Omron CX-Programmer project NewProject (CX-Programmer 9.61)

# PLC NewPLC1: CP1H XA

## Global symbols (name address type ; comment)
0.01 BOOL  ; Gr_out_up
0.02 BOOL  ; up_outside_1
0.03 BOOL  ; dn_outside_1
0.04 BOOL  ; dn_outside_2
0.05 BOOL  ; Gr_inside
0.06 BOOL  ; 1_inside
0.07 BOOL  ; 2_inside
100.01 BOOL  ; Motorup
100.02 BOOL  ; Motordown
100.03 BOOL  ; slow
100.04 BOOL  ; D_open
100.05 BOOL  ; D_close
100.09 BOOL  ; M111
10.00 BOOL  ; M1
10.01 BOOL  ; M2
10.02 BOOL  ; M3
10.03 BOOL  ; M4
10.04 BOOL  ; M5
10.05 BOOL  ; M3
10.06 BOOL  ; M7
10.07 BOOL  ; M8
10.08 BOOL  ; M9
10.09 BOOL  ; M10
10.10 BOOL  ; M11
10.11 BOOL  ; M12
10.12 BOOL  ; M13
10.13 BOOL  ; G_motor_up
10.14 BOOL  ; G_motorup_slow
10.15 BOOL  ; 1F_motor_up
11.01 BOOL  ; 1F_motor_slow
11.02 BOOL  ; 2F_motor_down
11.03 BOOL  ; 2F_motor_slow
11.04 BOOL  ; 1F_motor_down
11.05 BOOL  ; 1F_motor_slow
11.06 BOOL  ; G_motor_up_to_2nd
11.07 BOOL  ; G_motor_slow_to_2nd
11.08 BOOL  ; 2F_motor_down_toGround
11.09 BOOL  ; 2F_motor_slow_toGround
12.01 BOOL  ; 1F_pressed_slow
12.02 BOOL  ; 1F_pressed_stop
12.03 BOOL  ; 1F_pressed_slow1
12.04 BOOL  ; 1F_pressed_stopp
12.05 BOOL  ; M_2inside
12.06 BOOL  ; M_Ginside
13.01 BOOL  ; D_Open_for_outside
13.02 BOOL  ; D_Close_for_outside
13.03 BOOL  ; D_open_for_inside
13.04 BOOL  ; D_close_for_inside
13.05 BOOL  ; D_close_memory
13.06 BOOL  ; D_close_memory1
14.01 BOOL  ; MD1
14.02 BOOL  ; MD2
14.03 BOOL  ; MD3
14.04 BOOL  ; MD4
15.01 BOOL  ; M111
1.01 BOOL  ; LS0
1.02 BOOL  ; LS0(High)
1.03 BOOL  ; LS1
1.04 BOOL  ; LS1(High)
1.05 BOOL  ; LS2
1.06 BOOL  ; LS1(Low)
1.07 BOOL  ; LS0(Low)
T0000 BOOL  ; T1
T0001 BOOL  ; T2
T0002 BOOL  ; T3
T0003 BOOL  ; T4

## Program NewProgram1 (cyclic task 0)

### Section Section1

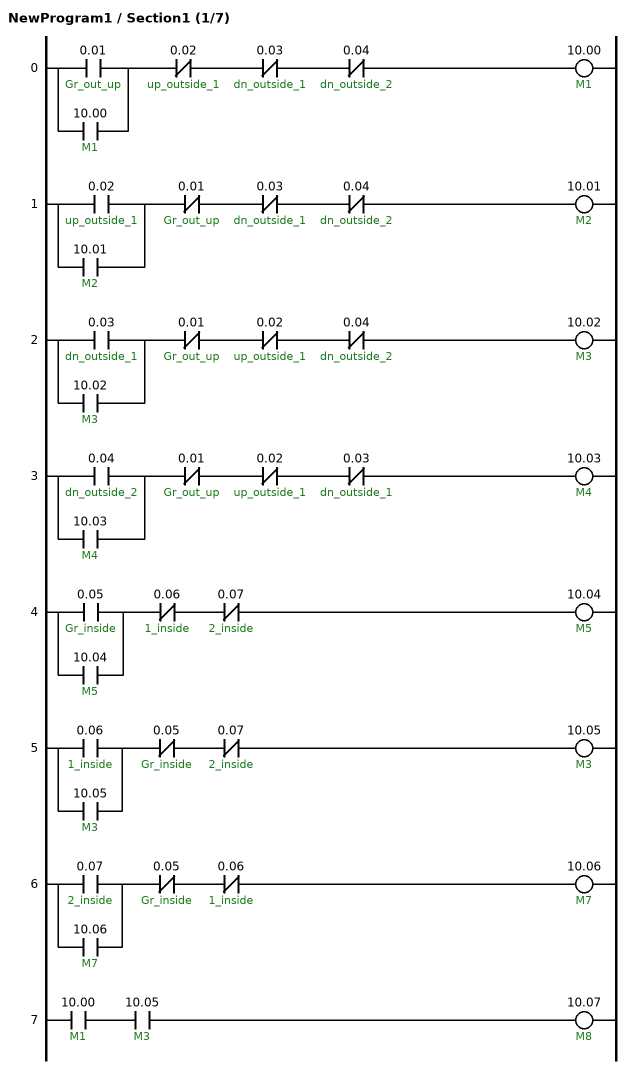
; rung 0
LD 0.01  ; Gr_out_up
OR 10.00  ; M1
ANDNOT 0.02  ; up_outside_1
ANDNOT 0.03  ; dn_outside_1
ANDNOT 0.04  ; dn_outside_2
OUT 10.00  ; M1
; rung 1
LD 0.02  ; up_outside_1
OR 10.01  ; M2
ANDNOT 0.01  ; Gr_out_up
ANDNOT 0.03  ; dn_outside_1
ANDNOT 0.04  ; dn_outside_2
OUT 10.01  ; M2
; rung 2
LD 0.03  ; dn_outside_1
OR 10.02  ; M3
ANDNOT 0.01  ; Gr_out_up
ANDNOT 0.02  ; up_outside_1
ANDNOT 0.04  ; dn_outside_2
OUT 10.02  ; M3
; rung 3
LD 0.04  ; dn_outside_2
OR 10.03  ; M4
ANDNOT 0.01  ; Gr_out_up
ANDNOT 0.02  ; up_outside_1
ANDNOT 0.03  ; dn_outside_1
OUT 10.03  ; M4
; rung 4
LD 0.05  ; Gr_inside
OR 10.04  ; M5
ANDNOT 0.06  ; 1_inside
ANDNOT 0.07  ; 2_inside
OUT 10.04  ; M5
; rung 5
LD 0.06  ; 1_inside
OR 10.05  ; M3
ANDNOT 0.05  ; Gr_inside
ANDNOT 0.07  ; 2_inside
OUT 10.05  ; M3
; rung 6
LD 0.07  ; 2_inside
OR 10.06  ; M7
ANDNOT 0.05  ; Gr_inside
ANDNOT 0.06  ; 1_inside
OUT 10.06  ; M7
; rung 7
LD 10.00  ; M1
AND 10.05  ; M3
OUT 10.07  ; M8

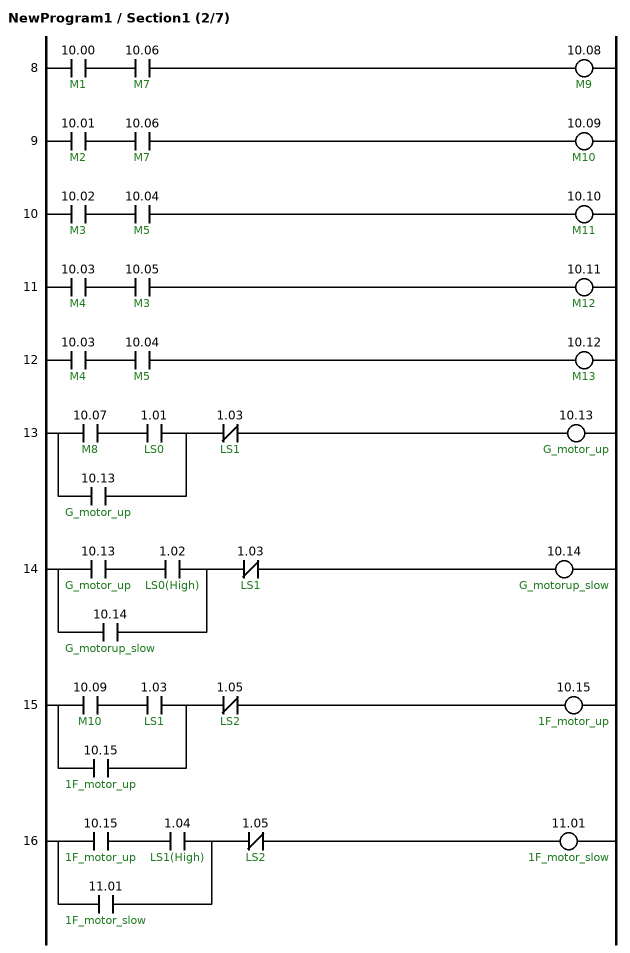
; rung 8
LD 10.00  ; M1
AND 10.06  ; M7
OUT 10.08  ; M9
; rung 9
LD 10.01  ; M2
AND 10.06  ; M7
OUT 10.09  ; M10
; rung 10
LD 10.02  ; M3
AND 10.04  ; M5
OUT 10.10  ; M11
; rung 11
LD 10.03  ; M4
AND 10.05  ; M3
OUT 10.11  ; M12
; rung 12
LD 10.03  ; M4
AND 10.04  ; M5
OUT 10.12  ; M13
; rung 13
LD 10.07  ; M8
AND 1.01  ; LS0
OR 10.13  ; G_motor_up
ANDNOT 1.03  ; LS1
OUT 10.13  ; G_motor_up
; rung 14
LD 10.13  ; G_motor_up
AND 1.02  ; LS0(High)
OR 10.14  ; G_motorup_slow
ANDNOT 1.03  ; LS1
OUT 10.14  ; G_motorup_slow
; rung 15
LD 10.09  ; M10
AND 1.03  ; LS1
OR 10.15  ; 1F_motor_up
ANDNOT 1.05  ; LS2
OUT 10.15  ; 1F_motor_up
; rung 16
LD 10.15  ; 1F_motor_up
AND 1.04  ; LS1(High)
OR 11.01  ; 1F_motor_slow
ANDNOT 1.05  ; LS2
OUT 11.01  ; 1F_motor_slow

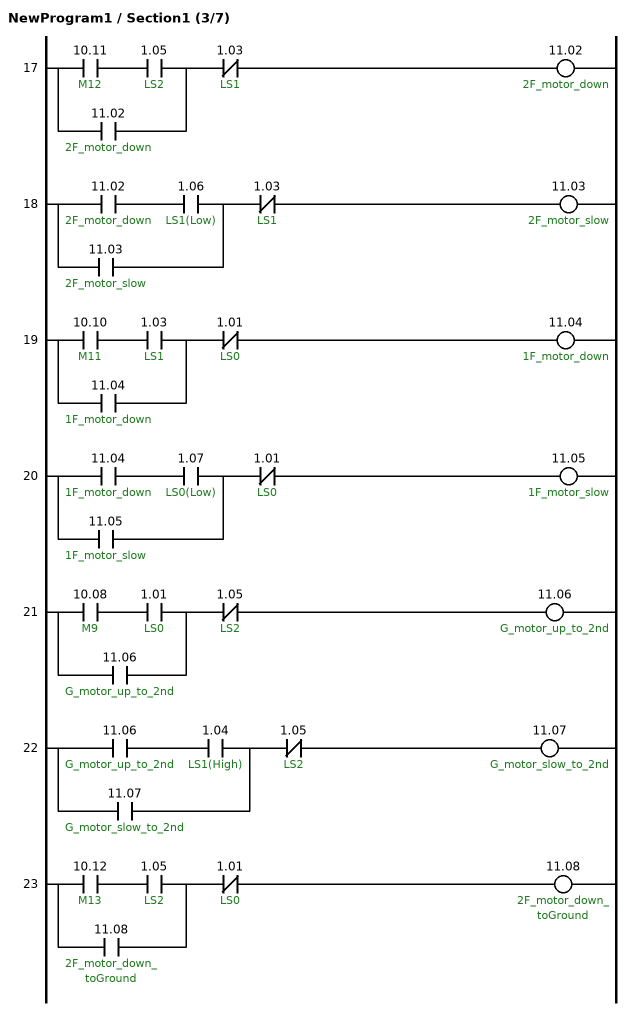
; rung 17
LD 10.11  ; M12
AND 1.05  ; LS2
OR 11.02  ; 2F_motor_down
ANDNOT 1.03  ; LS1
OUT 11.02  ; 2F_motor_down
; rung 18
LD 11.02  ; 2F_motor_down
AND 1.06  ; LS1(Low)
OR 11.03  ; 2F_motor_slow
ANDNOT 1.03  ; LS1
OUT 11.03  ; 2F_motor_slow
; rung 19
LD 10.10  ; M11
AND 1.03  ; LS1
OR 11.04  ; 1F_motor_down
ANDNOT 1.01  ; LS0
OUT 11.04  ; 1F_motor_down
; rung 20
LD 11.04  ; 1F_motor_down
AND 1.07  ; LS0(Low)
OR 11.05  ; 1F_motor_slow
ANDNOT 1.01  ; LS0
OUT 11.05  ; 1F_motor_slow
; rung 21
LD 10.08  ; M9
AND 1.01  ; LS0
OR 11.06  ; G_motor_up_to_2nd
ANDNOT 1.05  ; LS2
OUT 11.06  ; G_motor_up_to_2nd
; rung 22
LD 11.06  ; G_motor_up_to_2nd
AND 1.04  ; LS1(High)
OR 11.07  ; G_motor_slow_to_2nd
ANDNOT 1.05  ; LS2
OUT 11.07  ; G_motor_slow_to_2nd
; rung 23
LD 10.12  ; M13
AND 1.05  ; LS2
OR 11.08  ; 2F_motor_down_toGround
ANDNOT 1.01  ; LS0
OUT 11.08  ; 2F_motor_down_toGround

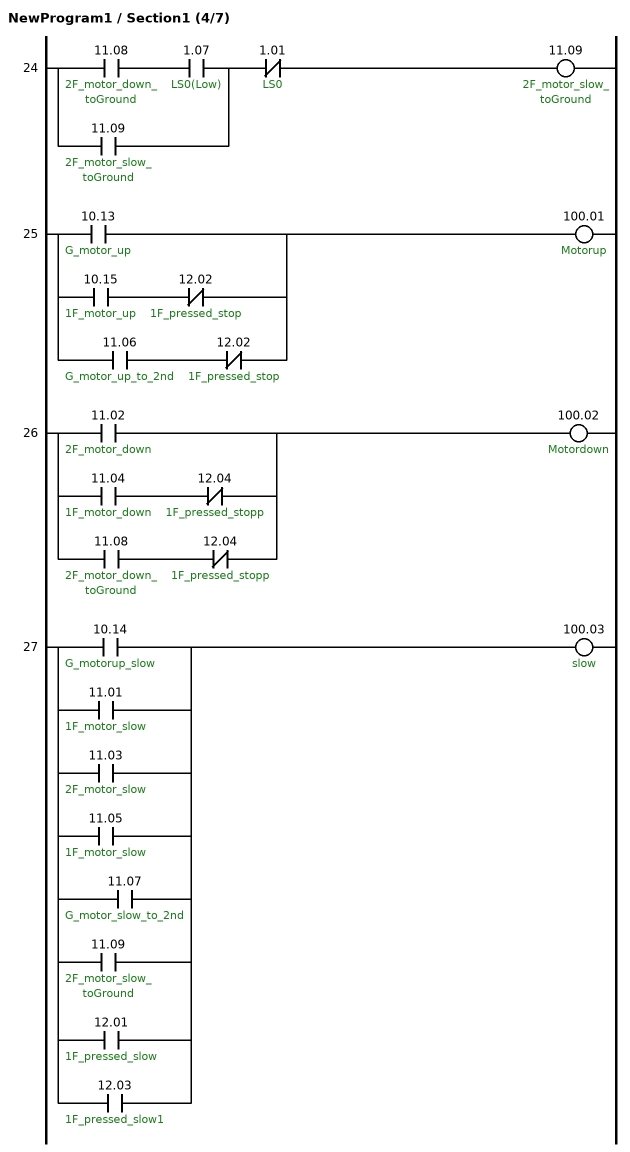
; rung 24
LD 11.08  ; 2F_motor_down_toGround
AND 1.07  ; LS0(Low)
OR 11.09  ; 2F_motor_slow_toGround
ANDNOT 1.01  ; LS0
OUT 11.09  ; 2F_motor_slow_toGround
; rung 25
LD 10.13  ; G_motor_up
LD 10.15  ; 1F_motor_up
ANDNOT 12.02  ; 1F_pressed_stop
ORLD
LD 11.06  ; G_motor_up_to_2nd
ANDNOT 12.02  ; 1F_pressed_stop
ORLD
OUT 100.01  ; Motorup
; rung 26
LD 11.02  ; 2F_motor_down
LD 11.04  ; 1F_motor_down
ANDNOT 12.04  ; 1F_pressed_stopp
ORLD
LD 11.08  ; 2F_motor_down_toGround
ANDNOT 12.04  ; 1F_pressed_stopp
ORLD
OUT 100.02  ; Motordown
; rung 27
LD 10.14  ; G_motorup_slow
OR 11.01  ; 1F_motor_slow
OR 11.03  ; 2F_motor_slow
OR 11.05  ; 1F_motor_slow
OR 11.07  ; G_motor_slow_to_2nd
OR 11.09  ; 2F_motor_slow_toGround
OR 12.01  ; 1F_pressed_slow
OR 12.03  ; 1F_pressed_slow1
OUT 100.03  ; slow

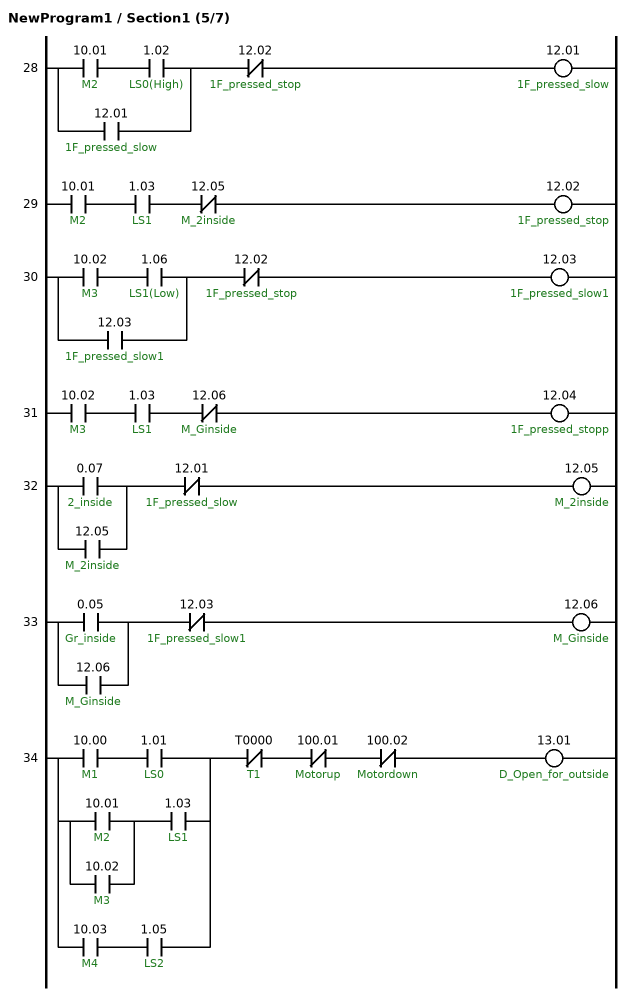
; rung 28
LD 10.01  ; M2
AND 1.02  ; LS0(High)
OR 12.01  ; 1F_pressed_slow
ANDNOT 12.02  ; 1F_pressed_stop
OUT 12.01  ; 1F_pressed_slow
; rung 29
LD 10.01  ; M2
AND 1.03  ; LS1
ANDNOT 12.05  ; M_2inside
OUT 12.02  ; 1F_pressed_stop
; rung 30
LD 10.02  ; M3
AND 1.06  ; LS1(Low)
OR 12.03  ; 1F_pressed_slow1
ANDNOT 12.02  ; 1F_pressed_stop
OUT 12.03  ; 1F_pressed_slow1
; rung 31
LD 10.02  ; M3
AND 1.03  ; LS1
ANDNOT 12.06  ; M_Ginside
OUT 12.04  ; 1F_pressed_stopp
; rung 32
LD 0.07  ; 2_inside
OR 12.05  ; M_2inside
ANDNOT 12.01  ; 1F_pressed_slow
OUT 12.05  ; M_2inside
; rung 33
LD 0.05  ; Gr_inside
OR 12.06  ; M_Ginside
ANDNOT 12.03  ; 1F_pressed_slow1
OUT 12.06  ; M_Ginside
; rung 34
LD 10.00  ; M1
AND 1.01  ; LS0
LD 10.01  ; M2
OR 10.02  ; M3
AND 1.03  ; LS1
ORLD
LD 10.03  ; M4
AND 1.05  ; LS2
ORLD
ANDNOT T0000  ; T1
ANDNOT 100.01  ; Motorup
ANDNOT 100.02  ; Motordown
OUT 13.01  ; D_Open_for_outside

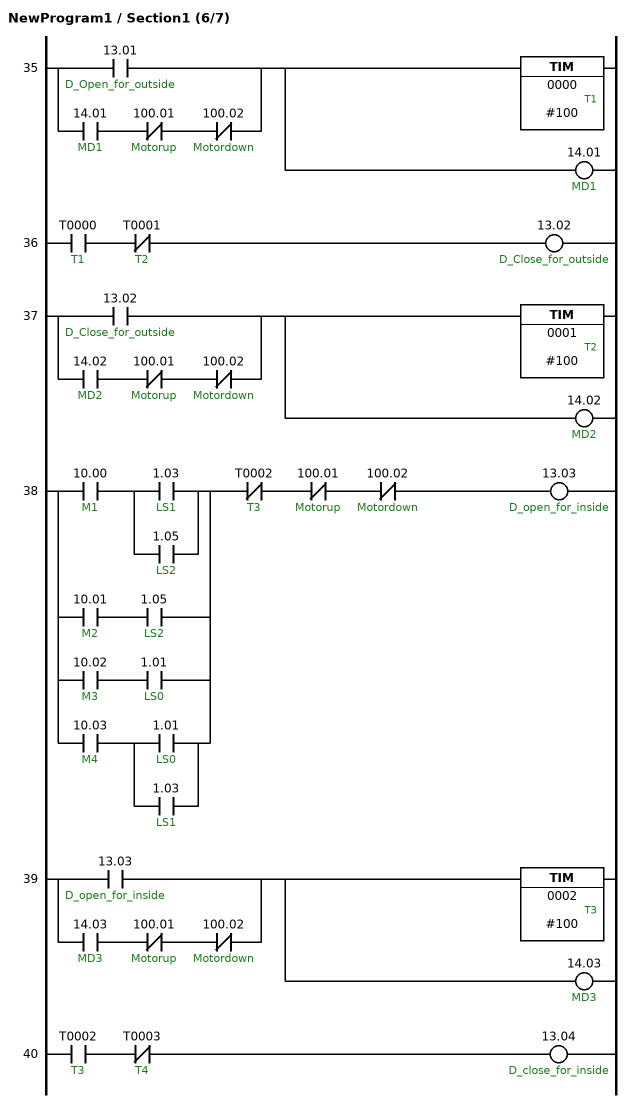
; rung 35
LD 13.01  ; D_Open_for_outside
LD 14.01  ; MD1
ANDNOT 100.01  ; Motorup
ANDNOT 100.02  ; Motordown
ORLD
TIM 0000 #100  ; T1
OUT 14.01  ; MD1
; rung 36
LD T0000  ; T1
ANDNOT T0001  ; T2
OUT 13.02  ; D_Close_for_outside
; rung 37
LD 13.02  ; D_Close_for_outside
LD 14.02  ; MD2
ANDNOT 100.01  ; Motorup
ANDNOT 100.02  ; Motordown
ORLD
TIM 0001 #100  ; T2
OUT 14.02  ; MD2
; rung 38
LD 10.00  ; M1
LD 1.03  ; LS1
OR 1.05  ; LS2
ANDLD
LD 10.01  ; M2
AND 1.05  ; LS2
ORLD
LD 10.02  ; M3
AND 1.01  ; LS0
ORLD
LD 10.03  ; M4
LD 1.01  ; LS0
OR 1.03  ; LS1
ANDLD
ORLD
ANDNOT T0002  ; T3
ANDNOT 100.01  ; Motorup
ANDNOT 100.02  ; Motordown
OUT 13.03  ; D_open_for_inside
; rung 39
LD 13.03  ; D_open_for_inside
LD 14.03  ; MD3
ANDNOT 100.01  ; Motorup
ANDNOT 100.02  ; Motordown
ORLD
TIM 0002 #100  ; T3
OUT 14.03  ; MD3
; rung 40
LD T0002  ; T3
ANDNOT T0003  ; T4
OUT 13.04  ; D_close_for_inside

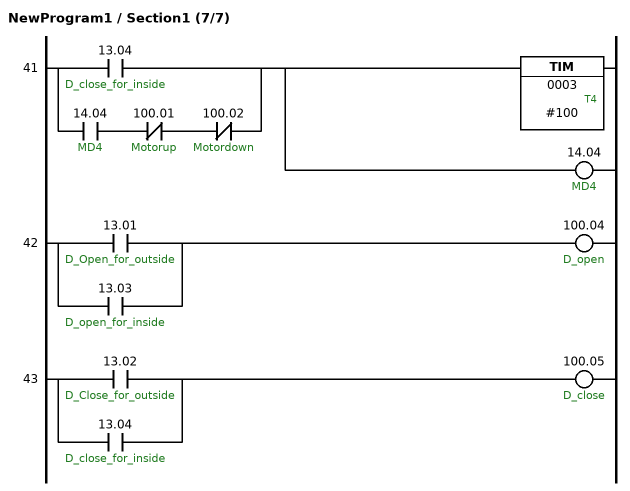
; rung 41
LD 13.04  ; D_close_for_inside
LD 14.04  ; MD4
ANDNOT 100.01  ; Motorup
ANDNOT 100.02  ; Motordown
ORLD
TIM 0003 #100  ; T4
OUT 14.04  ; MD4
; rung 42
LD 13.01  ; D_Open_for_outside
OR 13.03  ; D_open_for_inside
OUT 100.04  ; D_open
; rung 43
LD 13.02  ; D_Close_for_outside
OR 13.04  ; D_close_for_inside
OUT 100.05  ; D_close

### Section END
; rung 0
END(001)